TYPE NodeProfile :
STRUCT
	lastExecTime : LREAL;
	minExecTime : LREAL;
	maxExecTime : LREAL;
	averageExecTime : LREAL;
	measureCycle : DWORD;
END_STRUCT
END_TYPE

(* stored: Version 1.1.0.1, ProductVersion 3.1.4024.12
   DUT NodeProfile: Id {e4952ffa-5ad9-025f-30e0-08ac30e4e263} *)
